SYSTEM WORKER_HMI_Bachelor (* System Configuration *)
  (* Standard: 61499-1 *)
  (* Version 0.3, 2003-12-05, JHC, Rockwell Automation, Renamed from NEWSYSTEM. *)
  (* Version 0.2, 2002-11-05, JHC, Rockwell Automation, Fixed missing (empty) FBD in Application. *)
  (* Version 0.1, 2002-01-17, JHC, Rockwell Automation, Minor cleanup *)
  (* Version 0.0, 2000-05-27, JHC, Rockwell Automation *)
  APPLICATION APP1
  END_APPLICATION
  DEVICE WORKER_HMI_DEVICE : FRAME_DEVICE(BOUNDS := [1100,300,600,400], GRID := [1,1])
    RESOURCE WORKER_HMI_PROCESSOR : PANEL_RESOURCE(ROWS := 6, COLS := 2)
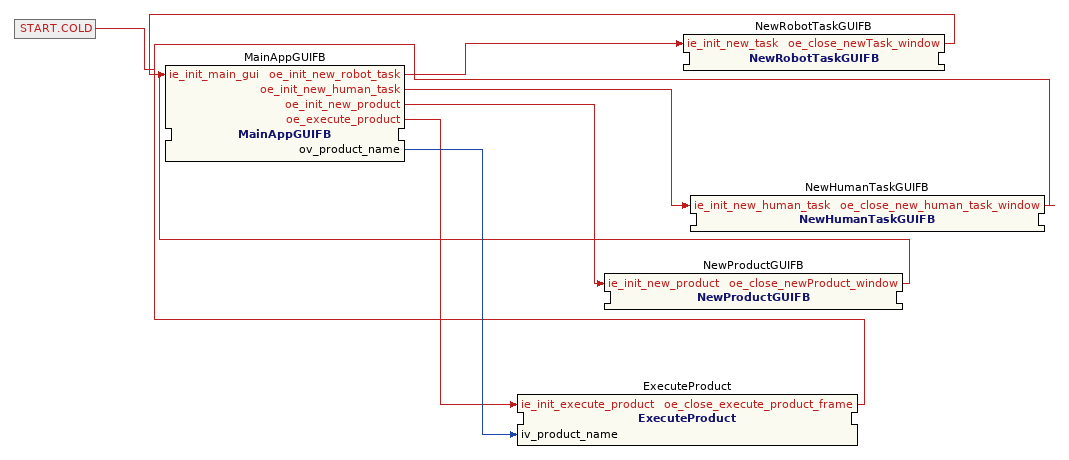
      FBS
        MainAppGUIFB : MainAppGUIFB;
        NewHumanTaskGUIFB : NewHumanTaskGUIFB;
        NewRobotTaskGUIFB : NewRobotTaskGUIFB;
        NewProductGUIFB : NewProductGUIFB;
        ExecuteProduct : ExecuteProduct;
      END_FBS
      EVENT_CONNECTIONS
        MainAppGUIFB.oe_init_new_robot_task TO NewRobotTaskGUIFB.ie_init_new_task;
        MainAppGUIFB.oe_init_new_human_task TO NewHumanTaskGUIFB.ie_init_new_human_task;
        MainAppGUIFB.oe_init_new_product TO NewProductGUIFB.ie_init_new_product;
        MainAppGUIFB.oe_execute_product TO ExecuteProduct.ie_init_execute_product;
        ExecuteProduct.oe_close_execute_product_frame TO MainAppGUIFB.ie_init_main_gui;
        NewProductGUIFB.oe_close_newProduct_window TO MainAppGUIFB.ie_init_main_gui;
        NewHumanTaskGUIFB.oe_close_new_human_task_window TO MainAppGUIFB.ie_init_main_gui;
        NewRobotTaskGUIFB.oe_close_newTask_window TO MainAppGUIFB.ie_init_main_gui;
        START.COLD TO MainAppGUIFB.ie_init_main_gui;
      END_CONNECTIONS
      DATA_CONNECTIONS
        MainAppGUIFB.ov_product_name TO ExecuteProduct.iv_product_name;
      END_CONNECTIONS
    END_RESOURCE
  END_DEVICE
END_SYSTEM
